// TIA Portal V18 export
ORGANIZATION_BLOCK "DevBlock"   // OB1, LAD, ProgramCycle
TITLE = "Main Program Sweep (Cycle)"
{ S7_Optimized_Access := 'TRUE' }
VERSION : 0.1
// stored: AutoNumber true, IsIECCheckEnabled false, SetENOAutomatically false
   VAR_INPUT
      Initial_Call : Bool;   // Initial call of this OB
      Remanence : Bool;   // =True, if remanent data are available
   END_VAR
   VAR_TEMP
      CappingStationTesting01 : Bool;
      CappingStationTesting02 : Bool;
      CappingStationTesting03 : Bool;
   END_VAR
BEGIN

REGION Network 1: Testing Capping Station
   // Use to perform cyclic test of the capping station.
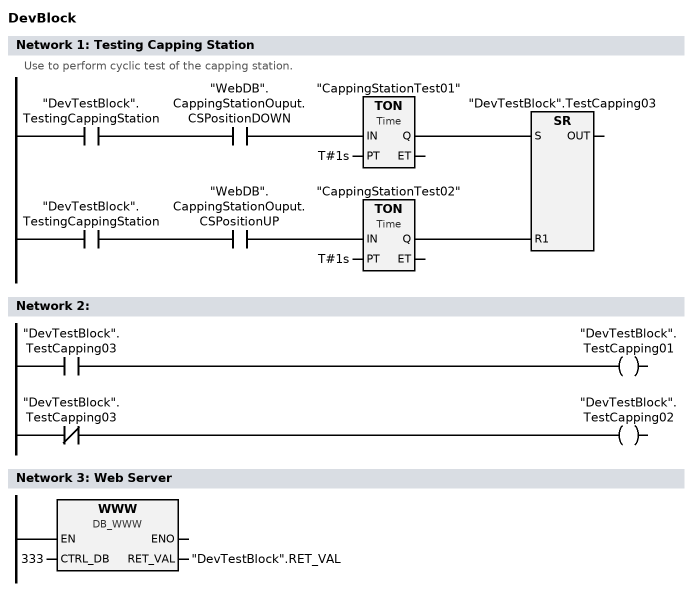
   RUNG wire#powerrail
      Contact( "DevTestBlock".TestingCappingStation )
      Contact( "WebDB".CappingStationOuput.CSPositionDOWN )
      { S7_Templates := "time_type := Time" } "CappingStationTest01".TON(pt := T#1s, et =>)
      S_SR(operand := "DevTestBlock".TestCapping03, r1 := wire#w1)
   END_RUNG
   RUNG wire#powerrail
      Contact( "DevTestBlock".TestingCappingStation )
      Contact( "WebDB".CappingStationOuput.CSPositionUP )
      { S7_Templates := "time_type := Time" } "CappingStationTest02".TON(pt := T#1s, et =>)
   END_RUNG wire#w1
   // the same network as SCL:
   "CappingStationTest01".TON(IN := "DevTestBlock".TestingCappingStation AND "WebDB".CappingStationOuput.CSPositionDOWN,
                           PT := T#1s);
   "CappingStationTest02".TON(IN := "DevTestBlock".TestingCappingStation AND "WebDB".CappingStationOuput.CSPositionUP,
                           PT := T#1s);
   IF "CappingStationTest01".Q THEN
       "DevTestBlock".TestCapping03 := TRUE;   // SR flip-flop
   END_IF;
   IF "CappingStationTest02".Q THEN "DevTestBlock".TestCapping03 := FALSE; END_IF;
END_REGION

REGION Network 2
   RUNG wire#powerrail
      Contact( "DevTestBlock".TestCapping03 )
      Coil( "DevTestBlock".TestCapping01 )
   END_RUNG
   RUNG wire#powerrail
      I_Contact( "DevTestBlock".TestCapping03 )
      Coil( "DevTestBlock".TestCapping02 )
   END_RUNG
   // the same network as SCL:
   "DevTestBlock".TestCapping01 := "DevTestBlock".TestCapping03;
   "DevTestBlock".TestCapping02 := NOT "DevTestBlock".TestCapping03;
END_REGION

REGION Network 3: Web Server
   RUNG wire#powerrail
      { S7_Templates := "value_type := DB_WWW" } WWW(CTRL_DB := 333, RET_VAL => "DevTestBlock".RET_VAL)
   END_RUNG
   // the same network as SCL:
   "DevTestBlock".RET_VAL := WWW(CTRL_DB := 333);
END_REGION
END_ORGANIZATION_BLOCK
